FUNCTION_BLOCK FB_Module_CoilHolder_Old IMPLEMENTS I_Module
VAR_INPUT
	bEnable			: BOOL;
END_VAR
VAR_OUTPUT
END_VAR
VAR
	Components		: ARRAY [0..9] OF I_Component;

	fbACmotor		: FB_Component_ACmotor;
	fbCoilLock		: FB_Component_SingleValve;
	fbReedLock		: FB_Component_ReedSwitch;
	fbReedUnlock	: FB_Component_ReedSwitch;
	
	fbIndexBit1		: FB_Component_InductiveSensor;
	fbIndexBit2		: FB_Component_InductiveSensor;
	fbIndexBit3		: FB_Component_InductiveSensor;
	fbIndexBit4		: FB_Component_InductiveSensor;
	fbIndexBit5		: FB_Component_InductiveSensor;
	fbIndexReady	: FB_Component_InductiveSensor;
	
	nIndex			: INT;
	idx				: INT;
END_VAR

IF bEnable THEN
	fbACmotor(
		bDeviceActive 	:= GVL.bLenze1Relay,
		sName			:= 'AC motor plate',
		bEnable			:= TRUE,
		bE1jog1			:= GVL.bLenze1JogBit1,
		bE2jog2			:= GVL.bLenze1JogBit2,
		bE3DCbrake		:= GVL.bLenze1InjectionBrake,
		eE4Direction	:= GVL.bLenze1Direction);
		
	fbCoilLock(
		sName 	:= 'Coil Lock',
		bEnable := TRUE,
		bOutput := GVL.bUnlockCoilHolder);
		
	fbReedLock(
		bRawSignal	:= GVL.bCoilHolderLocked,
		tDebounce	:= T#5MS,
		tTimeout	:= T#0S,
		sName		:= 'plate locked reed',
		bEnable		:= TRUE);
		
	fbReedUnlock(
		bRawSignal	:= GVL.bCoilHolderUnlocked,
		tDebounce	:= T#5MS,
		tTimeout	:= T#0S,
		sName		:= 'plate unlocked reed',
		bEnable		:= TRUE);
		
	fbIndexBit1(bRawSignal := GVL.bCoilHolderIndexBit1,
		tDebounce 	:= T#5MS,
		tTimeout	:= T#0S,
		sName		:= 'plate index 1',
		bEnable		:= TRUE);
		
	fbIndexBit2(bRawSignal := GVL.bCoilHolderIndexBit2,
		tDebounce 	:= T#5MS,
		tTimeout	:= T#0S,
		sName		:= 'plate index 2',
		bEnable		:= TRUE);
		
	fbIndexBit3(bRawSignal := GVL.bCoilHolderIndexBit3,
		tDebounce 	:= T#5MS,
		tTimeout	:= T#0S,
		sName		:= 'plate index 3',
		bEnable		:= TRUE);
		
	fbIndexBit4(bRawSignal := GVL.bCoilHolderIndexBit4,
		tDebounce 	:= T#5MS,
		tTimeout	:= T#0S,
		sName		:= 'plate index 4',
		bEnable		:= TRUE);
		
	fbIndexBit5(bRawSignal := GVL.bCoilHolderIndexBit5,
		tDebounce 	:= T#5MS,
		tTimeout	:= T#0S,
		sName		:= 'plate index 5',
		bEnable		:= TRUE);
		
	fbIndexReady(bRawSignal := GVL.bCoilHolderIndexReady,
		tDebounce 	:= T#5MS,
		tTimeout	:= T#0S,
		sName		:= 'plate index ready',
		bEnable		:= TRUE);

	Components[0] := fbACmotor;
	Components[1] := fbCoilLock;
	Components[2] := fbReedLock;
	Components[3] := fbReedUnlock;
	Components[4] := fbIndexBit1;
	Components[5] := fbIndexBit2;
	Components[6] := fbIndexBit3;
	Components[7] := fbIndexBit4;
	Components[8] := fbIndexBit5;
	Components[9] := fbIndexReady;
	
	FOR idx := 0 TO 9 DO
    	Components[idx].M_Start();
	END_FOR;
	
	// when index ready bit is triggered, convert index bits to integer
	IF fbIndexReady.bSensorActive THEN
		nIndex := 	TO_INT(SHL(TO_UINT(fbIndexBit5.bSensorActive), 4) OR
					SHL(TO_UINT(fbIndexBit4.bSensorActive), 3) OR
					SHL(TO_UINT(fbIndexBit3.bSensorActive), 2) OR
					SHL(TO_UINT(fbIndexBit2.bSensorActive), 1) OR
					(TO_UINT(fbIndexBit1.bSensorActive)));
	END_IF
END_IF

METHOD M_GoTo : BOOL
VAR_INPUT
	nTargetIndex	: INT;
END_VAR

VAR
	cwSteps: INT;
	target: INT;
	ccwSteps: INT;
	shortestDistance : INT;
END_VAR
IF fbReedUnlock.bSensorActive THEN
	IF nTargetIndex = nIndex THEN									// if target index is reached, turn off motor, lock plate and signal done
		fbACmotor.M_SetFreq(Frequency := E_LenzeJogFreq.F0FF);
		M_Lock();
		M_GoTo := TRUE;
		RETURN;
	END_IF
	
	cwSteps  := (nTargetIndex - nIndex + 24) MOD 24;				// calculate how much cw & ccw steps needed to go to target
	ccwSteps := (nIndex - nTargetIndex + 24) MOD 24;
	
	IF cwSteps <= ccwSteps THEN										// set direction for shortest path to target
		fbACmotor.M_SetDir(Direction := E_RotationDirection.CW);
		shortestDistance := cwSteps;
	ELSE
		fbACmotor.M_SetDir(Direction := E_RotationDirection.CCW);	
		shortestDistance := ccwSteps;
	END_IF
	
	IF nIndex <> nTargetIndex THEN
		IF shortestDistance <= 1 THEN								// if 1 from the target, set speed to slowest
			fbACmotor.M_SetFreq(Frequency := E_LenzeJogFreq.F1);	
		ELSIF shortestDistance <= 2 THEN							// if 2 from the target, set speed to slow
			fbACmotor.M_SetFreq(Frequency := E_LenzeJogFreq.F2);
		ELSE
			fbACmotor.M_SetFreq(Frequency := E_LenzeJogFreq.F3);	// if further set to highest speed
		END_IF
	ELSE
		fbACmotor.M_SetFreq(Frequency := E_LenzeJogFreq.F0FF);		// for safety, should be handled by first if
		M_Lock();
		M_GoTo := TRUE;
	END_IF
ELSE
	M_Unlock();														// unlock plate if locked
END_IF
END_METHOD

METHOD M_Halt : BOOL
VAR_INPUT
END_VAR
END_METHOD

METHOD M_Lock : BOOL
VAR_INPUT
END_VAR
fbCoilLock.M_Retract();
END_METHOD

METHOD M_Start : BOOL
VAR_INPUT
END_VAR
END_METHOD

METHOD M_Stop : BOOL
VAR_INPUT
END_VAR
END_METHOD

METHOD M_Unlock : BOOL
VAR_INPUT
END_VAR
fbCoilLock.M_Extend();
END_METHOD

END_FUNCTION_BLOCK

(* stored: Version 1.1.0.1, ProductVersion 3.1.4024.15
   POU FB_Module_CoilHolder_Old: Id {40d3fec2-1e88-465a-be78-81dbe38d536d}, SpecialFunc None
   Method M_GoTo: Id {17639c7b-edb3-4e9d-a3ae-83a1b7ed444e}
   Method M_Halt: Id {2d8dc12e-6061-4f13-b2a5-14d3305cde08}
   Method M_Lock: Id {cfd8b06a-dab1-4668-91c4-cb1bfb600106}
   Method M_Start: Id {c5a11795-bbe1-49cd-9dac-cdadbc4959da}
   Method M_Stop: Id {b19820e9-a53f-4b85-a742-f97acd7d8932}
   Method M_Unlock: Id {61de0c27-1f3d-4aac-a25b-a947746ff848} *)
